(* CODESYS project Library.library
   Version: 1.0.0.0
   Title: Tc3Build Library
   Placeholder: Tc3Build Library
   Company: Tc3Build

Project tree, tasks and I/O mapping:
  libraries: Tc2_Standard, * (Beckhoff Automation GmbH); Tc2_System, * (Beckhoff Automation GmbH)
  POUs/
    program MAIN [ST]
*)

// POUs/MAIN
PROGRAM MAIN
VAR
	_Count			: UINT;
END_VAR

_Count := _Count + 1;

END_PROGRAM
